INTERFACE I_FileFinder EXTENDS __SYSTEM.IQueryInterface

METHOD Find : BOOL;
VAR_INPUT
	SearchDirectory : T_MaxString;
	FileExtension : STRING;
END_VAR
END_METHOD

END_INTERFACE

(* stored: Version 1.1.0.1, ProductVersion 3.1.4024.9
   Itf I_FileFinder: Id {73be18f7-a4ad-4de2-a855-53f4ba6b8273}
   Method Find: Id {700e0810-b935-4015-aa88-7c7d02ab9009} *)
